// Mitsubishi GX Works2 project: sensor   PLC: Q02/Q02H

PROGRAM MAIN
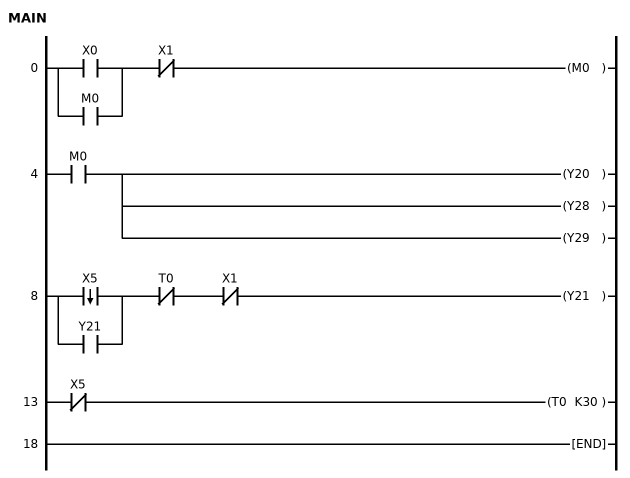
0     LD      X0
      OR      M0
      ANI     X1
      OUT     M0
4     LD      M0
      OUT     Y20
      OUT     Y28
      OUT     Y29
8     LDF     X5
      OR      Y21
      ANI     T0
      ANI     X1
      OUT     Y21
13    LDI     X5
      OUT     T0 K30
18    END
END_PROGRAM
